(* CODESYS project Einfacher_Fahrstuhl

Project tree, tasks and I/O mapping:
  Device : CODESYS Control Win V3 x64, CODESYS, version 3.5.20.10
    application Application
      libraries: Standard, 3.5.18.0 (System); Util, 3.5.19.0 (System)
      task MainTask (cyclic, interval 50 ms, priority 1, watchdog 100 ms x 4) calls Simulation, PLC_PRG
      task VISU_TASK (cyclic, interval 100 ms, priority 31) calls VisuElems.Visu_Prg
      function block DeactivateFloor [ST]
      global variables GVL
      function block NextFloor [ST]: FloorNumbers, GetNextBiggest, GetNextSmallest, Next
      program PLC_PRG [FBD]
      program Simulation [ST]
      visualisation Visualization
  libraries: VisuSymbols, 4.5.0.0 (System)
  text list GlobalTextList
*)

// Device/Application/GVL
VAR_GLOBAL
	FloorButtons			:	ARRAY [0..10] OF BOOL;
	CurrentElevatorFloor	:	BYTE;
	OnFloor					:	BOOL;
	AimedFloor				:	BYTE;
	
	CmdElevatorUp			:	BOOL;
	CmdElevatorDown			:	BOOL;
	
	NumberOfPressedFloors	:	BYTE;
	
END_VAR

// Device/Application/Simulation
PROGRAM Simulation
VAR
END_VAR
VAR_INPUT
	init : BOOL;
END_VAR

IF init = FALSE THEN
	CurrentElevatorFloor := 0;
	OnFloor := TRUE;
	
	
END_IF

END_PROGRAM

// Device/Application/PLC_PRG
PROGRAM PLC_PRG
VAR


	DeactivateFloor	:		DeactivateFloor;
	OffBoardDelay	:		TP;
	init			:		BOOL := FALSE;
	stopdelay		:		Ton;
	drivedelay		:		TOn;
	velocity		:		TIME := T#500MS;
	BLINK			:		BLINK;
	TaktUp			:		BLINK;
	TaktDown		:		BLINK;
	
	NextFloor		:		NextFloor;
	sr1				:		rs;
	sr2				:		rs;
	rtrig			:		R_TRIG;
	
	Upwards: BOOL;
	downwards: BOOL;

	FloorReached	:		R_TRIG;
	ButtonPressed	:		BOOL;

	
	FloorCounter	:		CTUD;
	TrueCounter		:		CTU;
	i				:		BYTE;
	StartingFloor	:		BYTE :=	CurrentElevatorFloor;
	

END_VAR
VAR // added by the converter: edge detectors and wires of the graphical bodies
    _w1, _w2 : BOOL;
END_VAR

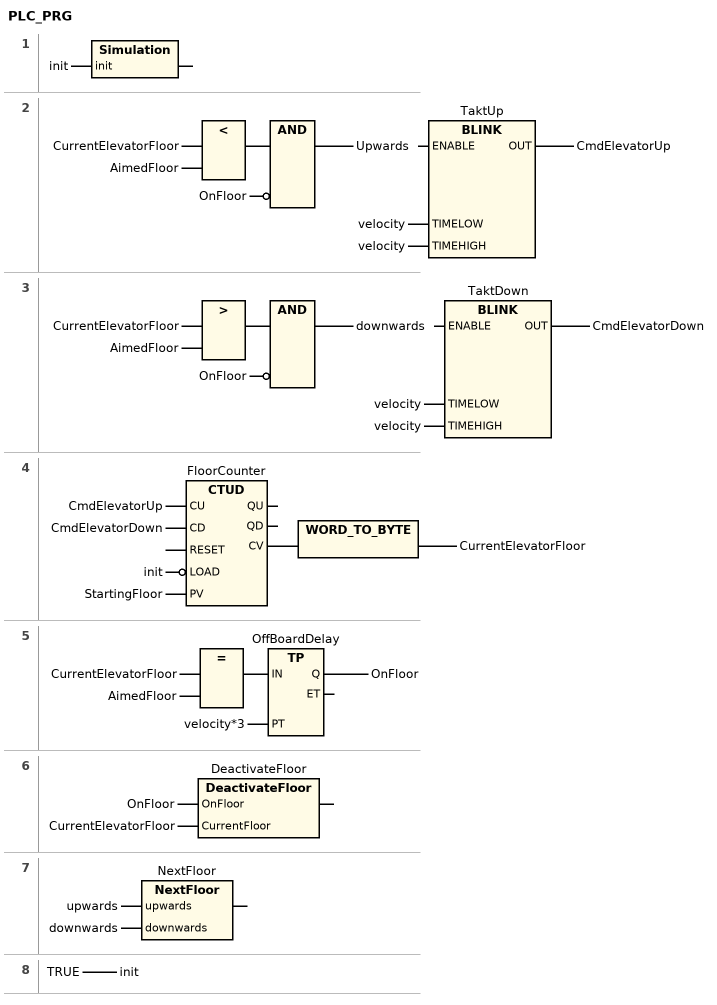
// NETWORK 1
Simulation(init := init);

// NETWORK 2
_w1 := CurrentElevatorFloor < AimedFloor AND NOT OnFloor;
Upwards := _w1;
TaktUp(ENABLE := _w1, TIMELOW := velocity, TIMEHIGH := velocity); // BLINK
CmdElevatorUp := TaktUp.OUT;

// NETWORK 3
_w2 := CurrentElevatorFloor > AimedFloor AND NOT OnFloor;
downwards := _w2;
TaktDown(ENABLE := _w2, TIMELOW := velocity, TIMEHIGH := velocity); // BLINK
CmdElevatorDown := TaktDown.OUT;

// NETWORK 4
FloorCounter(CU := CmdElevatorUp, CD := CmdElevatorDown, LOAD := NOT init, PV := StartingFloor); // CTUD
CurrentElevatorFloor := WORD_TO_BYTE(FloorCounter.CV);

// NETWORK 5
OffBoardDelay(IN := CurrentElevatorFloor = AimedFloor, PT := velocity*3); // TP
OnFloor := OffBoardDelay.Q;

// NETWORK 6
DeactivateFloor(OnFloor := OnFloor, CurrentFloor := CurrentElevatorFloor);

// NETWORK 7
NextFloor(upwards := upwards, downwards := downwards);

// NETWORK 8
init := TRUE;

END_PROGRAM

// Device/Application/DeactivateFloor
FUNCTION_BLOCK DeactivateFloor
VAR_INPUT
	OnFloor : BOOL;
	CurrentFloor : WORD;
END_VAR
VAR_OUTPUT
END_VAR
VAR
END_VAR

IF OnFloor = TRUE THEN
	FloorButtons[CurrentFloor] := FALSE;

END_IF

END_FUNCTION_BLOCK

// Device/Application/NextFloor
FUNCTION_BLOCK NextFloor
VAR_INPUT
	upwards:	BOOL;
	downwards: BOOL;
END_VAR
VAR_OUTPUT
END_VAR
VAR
	LastPosition:	BYTE;
	Buttons		:	ARRAY [0..10] OF BOOL;
	Floors		: 	BYTE;
	rs1			:	rs;
	rs2			:	rs;


	i			:	BYTE;
	BLINK		:	BLINK;
	GNS			:	BYTE;
	GNB			:	BYTE;

END_VAR

BLINK(ENABLE := TRUE, TIMELOW := T#100MS, TIMEHIGH := T#50MS);




IF BLINK.OUT OR OnFloor THEN
	Buttons := FloorButtons;
	
	Floors := FloorNumbers();
	IF Floors = 0 THEN
		AimedFloor := CurrentElevatorFloor;
	END_IF

	
	IF Floors = 1 THEN
		AimedFloor := Next();
	END_IF

	GNB := GetNextBiggest();
	IF (Floors > 1 AND CurrentElevatorFloor < 10 AND GNB <> 31 AND Upwards) OR (Floors> 1 AND CurrentElevatorFloor = 0) THEN
		GNB := GetNextBiggest();
		AimedFloor := GNB;
	END_IF
	
	GNS := GetNextSmallest();
	IF (Floors > 1 AND CurrentElevatorFloor > 0 AND GNS <> 31 AND downwards) OR (Floors> 1 AND CurrentElevatorFloor = 10) THEN
		GNS := GetNextSmallest();
		AimedFloor := GNS;
	END_IF
	
	
	
END_IF

METHOD FloorNumbers : BYTE;
VAR_INPUT
END_VAR
VAR
	i : BYTE;
	j : BYTE;
END_VAR
j := 0;
FOR i := 0 TO 10 BY 1 DO;
	IF Buttons[i] = TRUE THEN
		j := j+1;
	END_IF
	FloorNumbers := j;
END_FOR
END_METHOD

METHOD GetNextBiggest : BYTE
VAR_INPUT
END_VAR
FOR i := 0 TO 10 BY 1 DO;
	IF Buttons[CurrentElevatorFloor + i] = TRUE THEN
		GetNextBiggest := CurrentElevatorFloor + i;
		EXIT;
	END_IF
	IF CurrentElevatorFloor + i = 10 AND Buttons[CurrentElevatorFloor + i] = FALSE THEN
		GetNextBiggest := 31;
		EXIT;
	END_IF
END_FOR
END_METHOD

METHOD GetNextSmallest : BYTE
VAR_INPUT
END_VAR
FOR i := 0 TO 10 BY 1 DO;
	IF Buttons[CurrentElevatorFloor - i] = TRUE THEN
		GetNextSmallest := CurrentElevatorFloor -1;
		EXIT;
	END_IF
	IF CurrentElevatorFloor - i = 0 AND Buttons[CurrentElevatorFloor - i]=FALSE THEN
		GetNextSmallest := 31;
		EXIT;
	END_IF
END_FOR
END_METHOD

METHOD Next : BYTE
VAR_INPUT
END_VAR
FOR i := 0 TO 10 BY 1 DO
	IF Buttons[i] = TRUE THEN
		Next := i;	
	END_IF
END_FOR
END_METHOD

END_FUNCTION_BLOCK

// Device/Application/Visualization
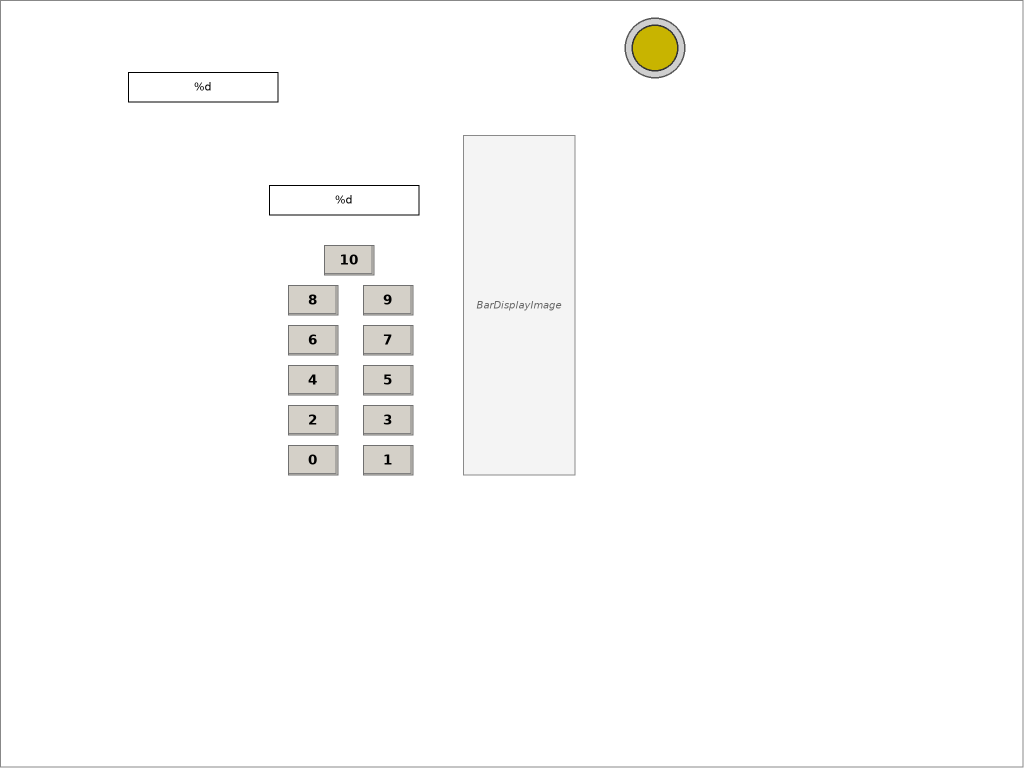
VISUALIZATION Visualization  // 1024x768
    Button (288,445 50x30), "0"
        toggle FloorButtons[0]
    Button (363,445 50x30), "1"
        toggle FloorButtons[1]
    Button (324,245 50x30), "10"
        toggle FloorButtons[10]
    Button (288,325 50x30), "6"
        toggle FloorButtons[6]
    Button (363,325 50x30), "7"
        toggle FloorButtons[7]
    Button (363,365 50x30), "5"
        toggle FloorButtons[5]
    Button (288,365 50x30), "4"
        toggle FloorButtons[4]
    Button (363,405 50x30), "3"
        toggle FloorButtons[3]
    Button (288,405 50x30), "2"
        toggle FloorButtons[2]
    Button (363,285 50x30), "9"
        toggle FloorButtons[9]
    Button (288,285 50x30), "8"
        toggle FloorButtons[8]
    BarDisplayImage (463,135 112x340), value: CurrentElevatorFloor, style: BarDisplayImage-Gray, scale format: %.1d, scale 0..10
    Rectangle (269,185 150x30), "%d", text variable: CurrentElevatorFloor
    Rectangle (128,72 150x30), "%d", text variable: NumberOfPressedFloors
    Lamp1 (620,13 70x70), variable: OnFloor, style: Lamp-Lamp1-Yellow
END_VISUALIZATION
